// TIA Portal project "Stanze_1" (V20)

(* hardware
DEVICE "S7-300/ET200M-Station_1"  S7-300 station
   slot 0: "Profilschiene_0"  Rail  6ES7 390-1***0-0AA0
   slot 2: "PLC_1"  CPU 315-2 PN/DP  6ES7 315-2EH14-0AB0  V3.2.18
      slot 2: "PROFINET-Schnittstelle_1"  PN-IO
         slot 1: "Port_1"  Port
         slot 2: "Port_2"  Port
   slot 4: "DI 16x24VDC_1"  DI16 x 24VDC, interrupt  6ES7 321-7BH01-0AB0
   slot 5: "DO 8x24VDC/0.5A_1"  DO8 x 24VDC / 0.5A  6ES7 322-8BF00-0AB0
*)

// ===== PLC "PLC_1"  CPU 315-2 PN/DP =====

VAR_GLOBAL   // PLC tag table "Standard-Variablentabelle"
   "Paketband_aktiv" AT %M1.0 : Bool;
   "Bauteil_erkannt" AT %M1.1 : Bool;
   "Paketband_stopppen" AT %M1.3 : Bool;
   "Stanze_aktivieren" AT %M3.0 : Bool;
   "Stanze_runter" AT %M3.1 : Bool;
   "Stanze_hoch" AT %M3.2 : Bool;
   "Stanzen_abgeschlossen" AT %M3.3 : Bool;
   "Stanze_oben" AT %M3.4 : Bool;
   "Start_freigeben" AT %M2.1 : Bool;
   "Bauteil_ausgerichtet" AT %M2.0 : Bool;
   "Paketband_verzögern" AT %M1.2 : Bool;
   "Start_sperren" AT %M1.4 : Bool;
   "Ausrichter_runter" AT %M2.2 : Bool;
END_VAR

VAR_GLOBAL   // PLC tag table "Eingänge"
   "S1" AT %I0.0 : Bool;   // Starttaster
   "B1" AT %I0.1 : Bool;   // Lichttaster
   "1b1" AT %I0.2 : Bool;   // Endlagensensor (Stanze)
   "1b2" AT %I0.3 : Bool;   // Stanzsensor
   "2b1" AT %E0.4 : Bool;   // Endlagensensor (Zange)
   "2b2" AT %E0.5 : Bool;   // Endlagensensor (Ausrichter)
END_VAR

VAR_GLOBAL   // PLC tag table "Ausgänge"
   "S1 (Licht)" AT %Q0.0 : Bool;   // Starttaster (Licht)
   "M1" AT %Q0.1 : Bool;   // Paketband
   "1Y1" AT %Q0.3 : Bool;   // Stanze
   "2Y1" AT %A0.4 : Bool;   // Ausrichter (Zange)
   "2Y2" AT %A0.5 : Bool;   // Ausrichter (Höhe)
END_VAR

FUNCTION "Stanzsteuerung" : Void   // FC1, FBD
{ S7_Optimized_Access := 'FALSE' }
VERSION : 0.1
   VAR_TEMP   // added for the SCL form of the ladder/FBD networks
      _w1 : Bool;
   END_VAR
BEGIN

REGION Network 1: Paketbandsteuerung (Start)
   // Mit drücken des S1 (Starttasters) wird das Paketband aktiviert, die Leuchte des Tasters leuchtet dann ebenfalls.
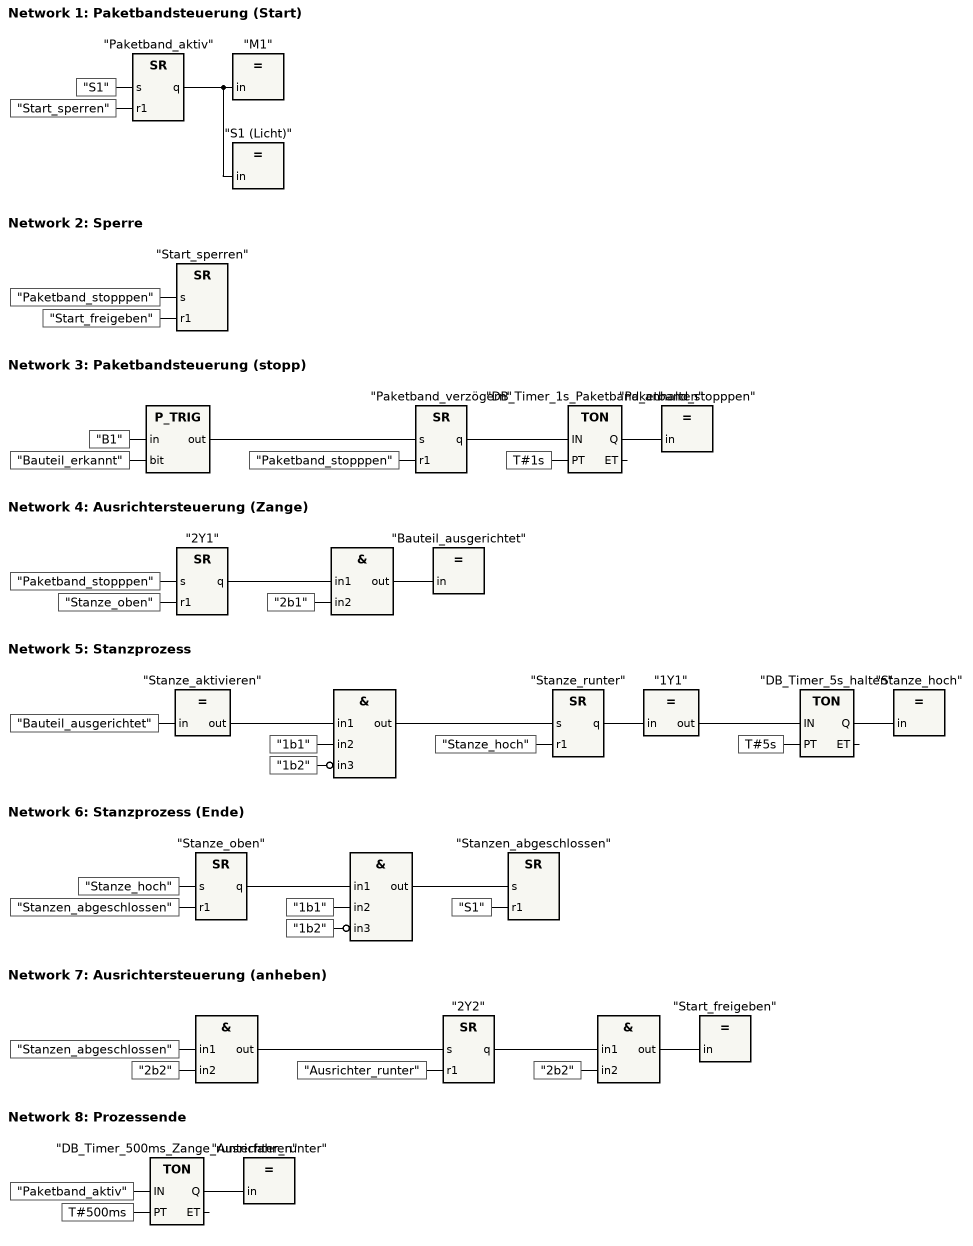
   IF "S1" THEN
       "Paketband_aktiv" := TRUE;   // SR flip-flop
   END_IF;
   IF "Start_sperren" THEN "Paketband_aktiv" := FALSE; END_IF;
   "M1" := "Paketband_aktiv";
   "S1 (Licht)" := "Paketband_aktiv";
END_REGION

REGION Network 2: Sperre
   // Das Band soll erst wieder gestartet werden, nachdem der Prozess abgeschlossen wurde.
   IF "Paketband_stopppen" THEN
       "Start_sperren" := TRUE;   // SR flip-flop
   END_IF;
   IF "Start_freigeben" THEN "Start_sperren" := FALSE; END_IF;
END_REGION

REGION Network 3: Paketbandsteuerung (stopp)
   // Nachdem der Sensor ein Bauteil erkennt, soll das Paketband nach ein paar Sekunden gestoppt werden. (Bis es den Ausrichter erreicht hat.)
   #_w1 := "B1" AND NOT "Bauteil_erkannt";   // rising edge
   "Bauteil_erkannt" := "B1";
   IF #_w1 THEN
       "Paketband_verzögern" := TRUE;   // SR flip-flop
   END_IF;
   IF "Paketband_stopppen" THEN "Paketband_verzögern" := FALSE; END_IF;
   "DB_Timer_1s_Paketband_anhalten".TON(IN := "Paketband_verzögern", PT := T#1s);
   "Paketband_stopppen" := "DB_Timer_1s_Paketband_anhalten".Q;
END_REGION

REGION Network 4: Ausrichtersteuerung (Zange)
   // Sobald das Paketband gestoppt ist (Bauteil hat Ausrichter erreicht), soll die Ausrichter-Zange das Bauteil festalten, bis der Stanzprozess abgeschlossen ist. Danach soll die Zange loslassen.
   IF "Paketband_stopppen" THEN
       "2Y1" := TRUE;   // SR flip-flop
   END_IF;
   IF "Stanze_oben" THEN "2Y1" := FALSE; END_IF;
   "Bauteil_ausgerichtet" := "2Y1" AND "2b1";
END_REGION

REGION Network 5: Stanzprozess
   // Sobald der Prozess gestartet wird, wird die Stanze runter gefahren und bleibt so lange unten, bis das Signal "Stanze_hoch" bekommt. Sobald die Stanze 5s angesteuert wurde, fährt die Stanze hoch.
   "Stanze_aktivieren" := "Bauteil_ausgerichtet";
   IF "Bauteil_ausgerichtet" AND "1b1" AND NOT "1b2" THEN
       "Stanze_runter" := TRUE;   // SR flip-flop
   END_IF;
   IF "Stanze_hoch" THEN "Stanze_runter" := FALSE; END_IF;
   "1Y1" := "Stanze_runter";
   "DB_Timer_5s_halten".TON(IN := "Stanze_runter", PT := T#5s);
   "Stanze_hoch" := "DB_Timer_5s_halten".Q;
END_REGION

REGION Network 6: Stanzprozess (Ende)
   // Nachdem die Stanze hoch gefahren ist, setze die anderen Flip-Flops zurück indem der Merker "Stanzen_abgeschlossen" gesetzt wird. Dieser kann mit drücken auf S1 (den Starttaster) zurück gesetzt werden.
   IF "Stanze_hoch" THEN
       "Stanze_oben" := TRUE;   // SR flip-flop
   END_IF;
   IF "Stanzen_abgeschlossen" THEN "Stanze_oben" := FALSE; END_IF;
   IF "Stanze_oben" AND "1b1" AND NOT "1b2" THEN
       "Stanzen_abgeschlossen" := TRUE;   // SR flip-flop
   END_IF;
   IF "S1" THEN "Stanzen_abgeschlossen" := FALSE; END_IF;
END_REGION

REGION Network 7: Ausrichtersteuerung (anheben)
   IF "Stanzen_abgeschlossen" AND "2b2" THEN
       "2Y2" := TRUE;   // SR flip-flop
   END_IF;
   IF "Ausrichter_runter" THEN "2Y2" := FALSE; END_IF;
   "Start_freigeben" := "2Y2" AND "2b2";
END_REGION

REGION Network 8: Prozessende
   // Nachdem das Paketband wieder gestartet wurde, fahre den Ausrichter 500 ms verzögert wieder nach unten.
   "DB_Timer_500ms_Zange_runterfahren".TON(IN := "Paketband_aktiv", PT := T#500ms);
   "Ausrichter_runter" := "DB_Timer_500ms_Zange_runterfahren".Q;
END_REGION
END_FUNCTION

ORGANIZATION_BLOCK "Main"   // OB1, FBD
TITLE = "Main Program Sweep (Cycle)"
{ S7_Optimized_Access := 'FALSE' }
VERSION : 0.1
   VAR_TEMP
      OB1_EV_CLASS : Byte;   // Bits 0-3 = 1 (Coming event), Bits 4-7 = 1 (Event class 1)
      OB1_SCAN_1 : Byte;   // 1 (Cold restart scan 1 of OB 1), 3 (Scan 2-n of OB 1)
      OB1_PRIORITY : Byte;   // Priority of OB Execution
      OB1_OB_NUMBR : Byte;   // 1 (Organization block 1, OB1)
      OB1_RESERVED_1 : Byte;   // Reserved for system
      OB1_RESERVED_2 : Byte;   // Reserved for system
      OB1_PREV_CYCLE : Int;   // Cycle time of previous OB1 scan (milliseconds)
      OB1_MIN_CYCLE : Int;   // Minimum cycle time of OB1 (milliseconds)
      OB1_MAX_CYCLE : Int;   // Maximum cycle time of OB1 (milliseconds)
      OB1_DATE_TIME : Date_And_Time;   // Date and time OB1 started
   END_VAR
BEGIN

REGION Network 1
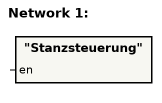
   "Stanzsteuerung"();
END_REGION
END_ORGANIZATION_BLOCK